(* PLC project cb_ctu, Dassault Systèmes ControlBuild 2024x *)
(* stored: creationDateTime 2023-10-03T11:12:45-01:00 *)

(* This is a IEC 1131-3 decounter. *)
FUNCTION_BLOCK timers_counters.cb_ctu
  VAR_INPUT
    CU : BOOL := false;
    R : BOOL := false;
    PV : INT := 0;
  END_VAR
  VAR_OUTPUT
    QU : BOOL := false;
    CV : INT := 0;
  END_VAR


ACTION C_source_code:
/* -----------------------------------------------------------------	*/
/* Type : BFU									*/
/* Copyright : Geensoft							*/
/* Version : 1.1 23/03/2010							*/
/* -----------------------------------------------------------------	*/
/* This is a Up-counter	  (CTU)					*/
/* -------------------------------------------------------------	*/
if(R) {
	CV = 0;
}
else {
	if(CU && (CV < 32767)) {
		CV  = CV  +1;
	}
}
QU =(CV >= PV);
END_ACTION
END_FUNCTION_BLOCK
